PROGRAM P_OutputNonCompensated
VAR
	fbValueInput 	: V2Q2u;
END_VAR

fbValueInput(
	Ps 	:= G_Sensors.fPressureSupply,
	Pa 	:= G_Sensors.fPressurePistonSide,
  	//Pa 	:= G_Simulator.fPistonSidePressure,
	Pb 	:= G_Sensors.fPressureRodSide,
  	//Pb 	:= G_Simulator.fRodSidePressure,
	y 	:= G_Sensors.fJoystickY,
	u	=> G_Work.fControlOutputNormalized
);

END_PROGRAM

(* stored: Version 1.1.0.1, ProductVersion 3.1.4024.12
   POU P_OutputNonCompensated: Id {91e8730f-330f-4841-8441-0d9eae6d44e6}, SpecialFunc None *)
